// Provides time information for an alarm
TYPE ST_AlarmTimeInfos :
STRUCT
	Activated		: Tc2_Utilities.TIMESTRUCT;	// Time of alarm activation
	Deactivated		: Tc2_Utilities.TIMESTRUCT;	// Time of alarm deactiovation
	Acknowledged	: Tc2_Utilities.TIMESTRUCT;	// Time of alarm acknowlidgemenet
END_STRUCT
END_TYPE

(* stored: Version 1.1.0.1
   DUT ST_AlarmTimeInfos: Id {d6222138-e632-0fde-0530-505c32c5c78b} *)
